// TIA Portal V16 export
// export: Created 2021-12-01T20:36:48.810046Z, ExportSetting WithDefaults, DisplayName Totally Integrated Automation Portal, DisplayVersion V16 Update 4, DisplayName TIA Portal Version Control Interface, DisplayVersion V16 Update 2, DisplayName TIA Portal Openness, DisplayVersion V16 Update 4, DisplayName SINAMICS Startdrive Advanced, DisplayVersion V16 Update 5, DisplayName SINAMICS Startdrive G130, G150, S120, S150, SINAMICS MV, S210, DisplayVersion V16 Update 5, DisplayName SINAMICS Startdrive G110M, G120, G120C, G120D, G120P, G115D, DisplayVersion V16 Update 5, DisplayName STEP 7 Professional, DisplayVersion V16 Update 4, DisplayName STEP 7 Safety, DisplayVersion V16, DisplayName WinCC Advanced, DisplayVersion V16 Update 4
FUNCTION "ST00280_FC" : Void   // FC102, LAD
TITLE = ST00280
{ S7_Optimized_Access := 'TRUE' }
VERSION : 0.1
// stored: AutoNumber true, IsIECCheckEnabled false, SetENOAutomatically false, UDAEnableTagReadback false
   VAR_IN_OUT
      OPMODE : "OPMODE_OUT_UDT";
      HMI_EXTENSION : "HMI_EXTENSION_PANEL_UDT";
   END_VAR
   VAR_TEMP
      EmptyHS : "RT_HANDSHAKE_UDT";
   END_VAR
BEGIN

REGION Network 1: Alarm
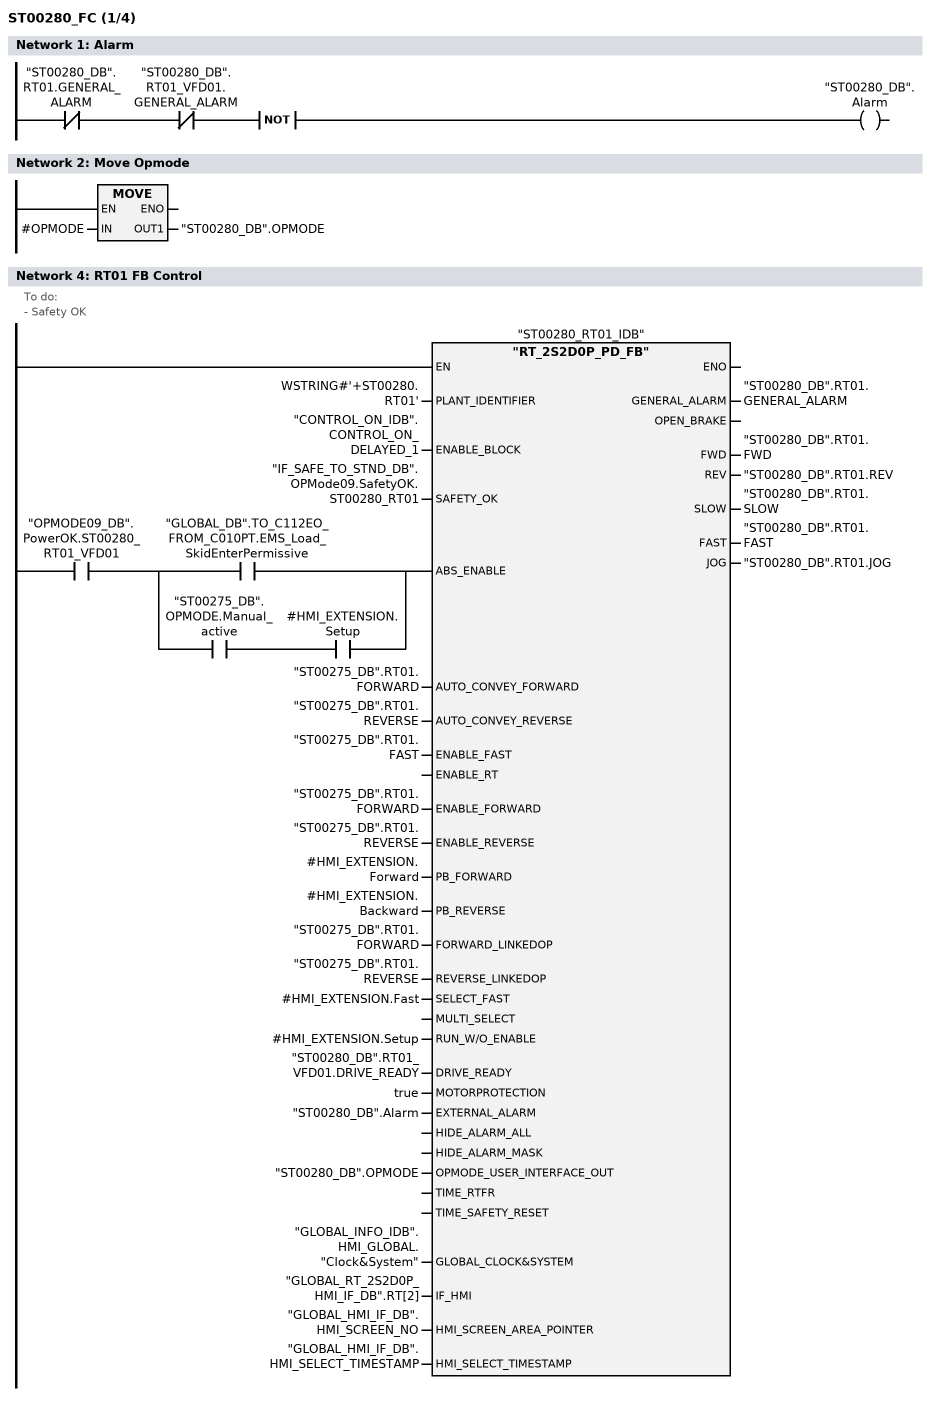
   RUNG wire#powerrail
      I_Contact( "ST00280_DB".RT01.GENERAL_ALARM )
      I_Contact( "ST00280_DB".RT01_VFD01.GENERAL_ALARM )
      Not()
      Coil( "ST00280_DB".Alarm )
   END_RUNG
   // the same network as SCL:
   "ST00280_DB".Alarm := NOT (NOT "ST00280_DB".RT01.GENERAL_ALARM AND NOT "ST00280_DB".RT01_VFD01.GENERAL_ALARM);
END_REGION

REGION Network 2: Move Opmode
   RUNG wire#powerrail
      Move(in := #OPMODE, out1 => "ST00280_DB".OPMODE)
   END_RUNG
   // the same network as SCL:
   "ST00280_DB".OPMODE := #OPMODE;
END_REGION

REGION Network 3: *******************RT01 Control*******************
END_REGION

REGION Network 4: RT01 FB Control
   // To do:
   // 										- Safety OK
   RUNG wire#powerrail
      "ST00280_RT01_IDB"(ABS_ENABLE := wire#w2, PLANT_IDENTIFIER := WSTRING#'+ST00280.RT01', ENABLE_BLOCK := "CONTROL_ON_IDB".CONTROL_ON_DELAYED_1, SAFETY_OK := "IF_SAFE_TO_STND_DB".OPMode09.SafetyOK.ST00280_RT01, AUTO_CONVEY_FORWARD := "ST00275_DB".RT01.FORWARD, AUTO_CONVEY_REVERSE := "ST00275_DB".RT01.REVERSE, ENABLE_FAST := "ST00275_DB".RT01.FAST, ENABLE_RT :=, ENABLE_FORWARD := "ST00275_DB".RT01.FORWARD, ENABLE_REVERSE := "ST00275_DB".RT01.REVERSE, PB_FORWARD := #HMI_EXTENSION.Forward, PB_REVERSE := #HMI_EXTENSION.Backward, FORWARD_LINKEDOP := "ST00275_DB".RT01.FORWARD, REVERSE_LINKEDOP := "ST00275_DB".RT01.REVERSE, SELECT_FAST := #HMI_EXTENSION.Fast, MULTI_SELECT :=, "RUN_W/O_ENABLE" := #HMI_EXTENSION.Setup, DRIVE_READY := "ST00280_DB".RT01_VFD01.DRIVE_READY, MOTORPROTECTION := true, EXTERNAL_ALARM := "ST00280_DB".Alarm, HIDE_ALARM_ALL :=, HIDE_ALARM_MASK :=, OPMODE_USER_INTERFACE_OUT := "ST00280_DB".OPMODE, TIME_RTFR :=, TIME_SAFETY_RESET :=, "GLOBAL_CLOCK&SYSTEM" := "GLOBAL_INFO_IDB".HMI_GLOBAL."Clock&System", IF_HMI := "GLOBAL_RT_2S2D0P_HMI_IF_DB".RT[2], HMI_SCREEN_AREA_POINTER := "GLOBAL_HMI_IF_DB".HMI_SCREEN_NO, HMI_SELECT_TIMESTAMP := "GLOBAL_HMI_IF_DB".HMI_SELECT_TIMESTAMP, GENERAL_ALARM => "ST00280_DB".RT01.GENERAL_ALARM, OPEN_BRAKE =>, FWD => "ST00280_DB".RT01.FWD, REV => "ST00280_DB".RT01.REV, SLOW => "ST00280_DB".RT01.SLOW, FAST => "ST00280_DB".RT01.FAST, JOG => "ST00280_DB".RT01.JOG)
   END_RUNG
   RUNG wire#powerrail
      Contact( "OPMODE09_DB".PowerOK.ST00280_RT01_VFD01 )
      wire#w1
      Contact( "GLOBAL_DB".TO_C112EO_FROM_C010PT.EMS_Load_SkidEnterPermissive )
   END_RUNG wire#w2
   RUNG wire#w1
      Contact( "ST00275_DB".OPMODE.Manual_active )
      Contact( #HMI_EXTENSION.Setup )
   END_RUNG wire#w2
   // the same network as SCL:
   "ST00280_RT01_IDB"(PLANT_IDENTIFIER := WSTRING#'+ST00280.RT01',   // "RT_2S2D0P_PD_FB"
                      ENABLE_BLOCK := "CONTROL_ON_IDB".CONTROL_ON_DELAYED_1,
                      SAFETY_OK := "IF_SAFE_TO_STND_DB".OPMode09.SafetyOK.ST00280_RT01,
                      ABS_ENABLE := "OPMODE09_DB".PowerOK.ST00280_RT01_VFD01 AND ("GLOBAL_DB".TO_C112EO_FROM_C010PT.EMS_Load_SkidEnterPermissive OR ("ST00275_DB".OPMODE.Manual_active AND #HMI_EXTENSION.Setup)),
                      AUTO_CONVEY_FORWARD := "ST00275_DB".RT01.FORWARD,
                      AUTO_CONVEY_REVERSE := "ST00275_DB".RT01.REVERSE,
                      ENABLE_FAST := "ST00275_DB".RT01.FAST,
                      ENABLE_FORWARD := "ST00275_DB".RT01.FORWARD,
                      ENABLE_REVERSE := "ST00275_DB".RT01.REVERSE,
                      PB_FORWARD := #HMI_EXTENSION.Forward,
                      PB_REVERSE := #HMI_EXTENSION.Backward,
                      FORWARD_LINKEDOP := "ST00275_DB".RT01.FORWARD,
                      REVERSE_LINKEDOP := "ST00275_DB".RT01.REVERSE,
                      SELECT_FAST := #HMI_EXTENSION.Fast,
                      "RUN_W/O_ENABLE" := #HMI_EXTENSION.Setup,
                      DRIVE_READY := "ST00280_DB".RT01_VFD01.DRIVE_READY,
                      MOTORPROTECTION := true,
                      EXTERNAL_ALARM := "ST00280_DB".Alarm,
                      OPMODE_USER_INTERFACE_OUT := "ST00280_DB".OPMODE,
                      "GLOBAL_CLOCK&SYSTEM" := "GLOBAL_INFO_IDB".HMI_GLOBAL."Clock&System",
                      IF_HMI := "GLOBAL_RT_2S2D0P_HMI_IF_DB".RT[2],
                      HMI_SCREEN_AREA_POINTER := "GLOBAL_HMI_IF_DB".HMI_SCREEN_NO,
                      HMI_SELECT_TIMESTAMP := "GLOBAL_HMI_IF_DB".HMI_SELECT_TIMESTAMP,
                      GENERAL_ALARM => "ST00280_DB".RT01.GENERAL_ALARM,
                      FWD => "ST00280_DB".RT01.FWD,
                      REV => "ST00280_DB".RT01.REV,
                      SLOW => "ST00280_DB".RT01.SLOW,
                      FAST => "ST00280_DB".RT01.FAST,
                      JOG => "ST00280_DB".RT01.JOG);
END_REGION

REGION Network 5: RT01 Speed
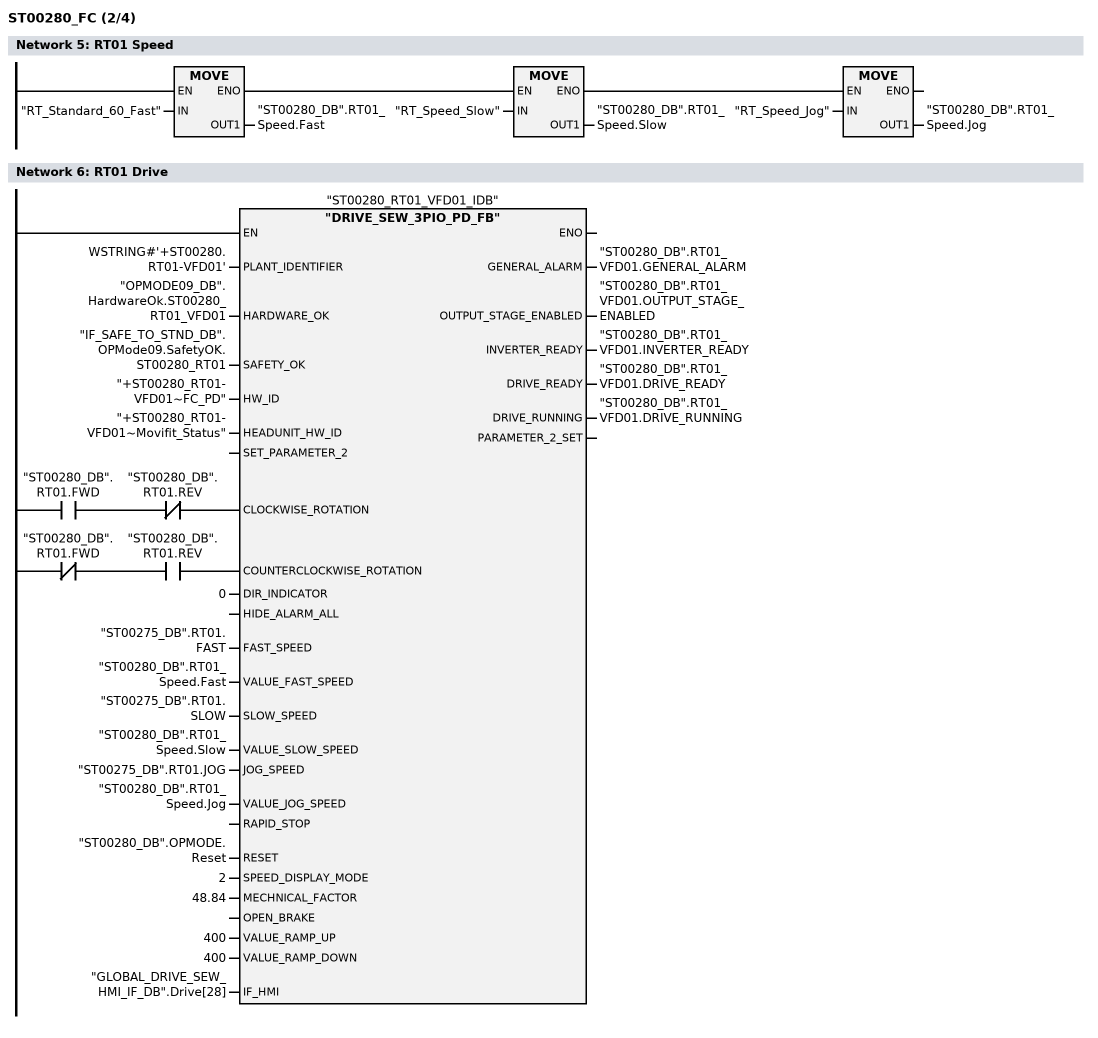
   RUNG wire#powerrail
      Move(in := "RT_Standard_60_Fast", out1 => "ST00280_DB".RT01_Speed.Fast)
      Move(in := "RT_Speed_Slow", out1 => "ST00280_DB".RT01_Speed.Slow)
      Move(in := "RT_Speed_Jog", out1 => "ST00280_DB".RT01_Speed.Jog)
   END_RUNG
   // the same network as SCL:
   "ST00280_DB".RT01_Speed.Fast := "RT_Standard_60_Fast";
   "ST00280_DB".RT01_Speed.Slow := "RT_Speed_Slow";
   "ST00280_DB".RT01_Speed.Jog := "RT_Speed_Jog";
END_REGION

REGION Network 6: RT01 Drive
   RUNG wire#powerrail
      "ST00280_RT01_VFD01_IDB"(CLOCKWISE_ROTATION := wire#w1, COUNTERCLOCKWISE_ROTATION := wire#w2, PLANT_IDENTIFIER := WSTRING#'+ST00280.RT01-VFD01', HARDWARE_OK := "OPMODE09_DB".HardwareOk.ST00280_RT01_VFD01, SAFETY_OK := "IF_SAFE_TO_STND_DB".OPMode09.SafetyOK.ST00280_RT01, HW_ID := "+ST00280_RT01-VFD01~FC_PD", HEADUNIT_HW_ID := "+ST00280_RT01-VFD01~Movifit_Status", SET_PARAMETER_2 :=, DIR_INDICATOR := 0, HIDE_ALARM_ALL :=, FAST_SPEED := "ST00275_DB".RT01.FAST, VALUE_FAST_SPEED := "ST00280_DB".RT01_Speed.Fast, SLOW_SPEED := "ST00275_DB".RT01.SLOW, VALUE_SLOW_SPEED := "ST00280_DB".RT01_Speed.Slow, JOG_SPEED := "ST00275_DB".RT01.JOG, VALUE_JOG_SPEED := "ST00280_DB".RT01_Speed.Jog, RAPID_STOP :=, RESET := "ST00280_DB".OPMODE.Reset, SPEED_DISPLAY_MODE := 2, MECHNICAL_FACTOR := 48.84, OPEN_BRAKE :=, VALUE_RAMP_UP := 400, VALUE_RAMP_DOWN := 400, IF_HMI := "GLOBAL_DRIVE_SEW_HMI_IF_DB".Drive[28], GENERAL_ALARM => "ST00280_DB".RT01_VFD01.GENERAL_ALARM, OUTPUT_STAGE_ENABLED => "ST00280_DB".RT01_VFD01.OUTPUT_STAGE_ENABLED, INVERTER_READY => "ST00280_DB".RT01_VFD01.INVERTER_READY, DRIVE_READY => "ST00280_DB".RT01_VFD01.DRIVE_READY, DRIVE_RUNNING => "ST00280_DB".RT01_VFD01.DRIVE_RUNNING, PARAMETER_2_SET =>)
   END_RUNG
   RUNG wire#powerrail
      Contact( "ST00280_DB".RT01.FWD )
      I_Contact( "ST00280_DB".RT01.REV )
   END_RUNG wire#w1
   RUNG wire#powerrail
      I_Contact( "ST00280_DB".RT01.FWD )
      Contact( "ST00280_DB".RT01.REV )
   END_RUNG wire#w2
   // the same network as SCL:
   "ST00280_RT01_VFD01_IDB"(PLANT_IDENTIFIER := WSTRING#'+ST00280.RT01-VFD01',   // "DRIVE_SEW_3PIO_PD_FB"
                           HARDWARE_OK := "OPMODE09_DB".HardwareOk.ST00280_RT01_VFD01,
                           SAFETY_OK := "IF_SAFE_TO_STND_DB".OPMode09.SafetyOK.ST00280_RT01,
                           HW_ID := "+ST00280_RT01-VFD01~FC_PD",
                           HEADUNIT_HW_ID := "+ST00280_RT01-VFD01~Movifit_Status",
                           CLOCKWISE_ROTATION := "ST00280_DB".RT01.FWD AND NOT "ST00280_DB".RT01.REV,
                           COUNTERCLOCKWISE_ROTATION := NOT "ST00280_DB".RT01.FWD AND "ST00280_DB".RT01.REV,
                           DIR_INDICATOR := 0,
                           FAST_SPEED := "ST00275_DB".RT01.FAST,
                           VALUE_FAST_SPEED := "ST00280_DB".RT01_Speed.Fast,
                           SLOW_SPEED := "ST00275_DB".RT01.SLOW,
                           VALUE_SLOW_SPEED := "ST00280_DB".RT01_Speed.Slow,
                           JOG_SPEED := "ST00275_DB".RT01.JOG,
                           VALUE_JOG_SPEED := "ST00280_DB".RT01_Speed.Jog,
                           RESET := "ST00280_DB".OPMODE.Reset,
                           SPEED_DISPLAY_MODE := 2,
                           MECHNICAL_FACTOR := 48.84,
                           VALUE_RAMP_UP := 400,
                           VALUE_RAMP_DOWN := 400,
                           IF_HMI := "GLOBAL_DRIVE_SEW_HMI_IF_DB".Drive[28],
                           GENERAL_ALARM => "ST00280_DB".RT01_VFD01.GENERAL_ALARM,
                           OUTPUT_STAGE_ENABLED => "ST00280_DB".RT01_VFD01.OUTPUT_STAGE_ENABLED,
                           INVERTER_READY => "ST00280_DB".RT01_VFD01.INVERTER_READY,
                           DRIVE_READY => "ST00280_DB".RT01_VFD01.DRIVE_READY,
                           DRIVE_RUNNING => "ST00280_DB".RT01_VFD01.DRIVE_RUNNING);
END_REGION

REGION Network 7: *******************PO01 Control*******************
END_REGION

REGION Network 8 (SCL): PO01 Parameters
   "ST00280_DB".PO01.PARA_SET.Para.PosEndForward2 := false;
   "ST00280_DB".PO01.PARA_SET.Para.PosEndReverse2 := false;

   "ST00280_DB".PO01.PARA_SET.Set.SetRT := 100;
   "ST00280_DB".PO01.PARA_SET.Set.TimePosLeft := 10;
END_REGION

REGION Network 9: PO01 FB Control
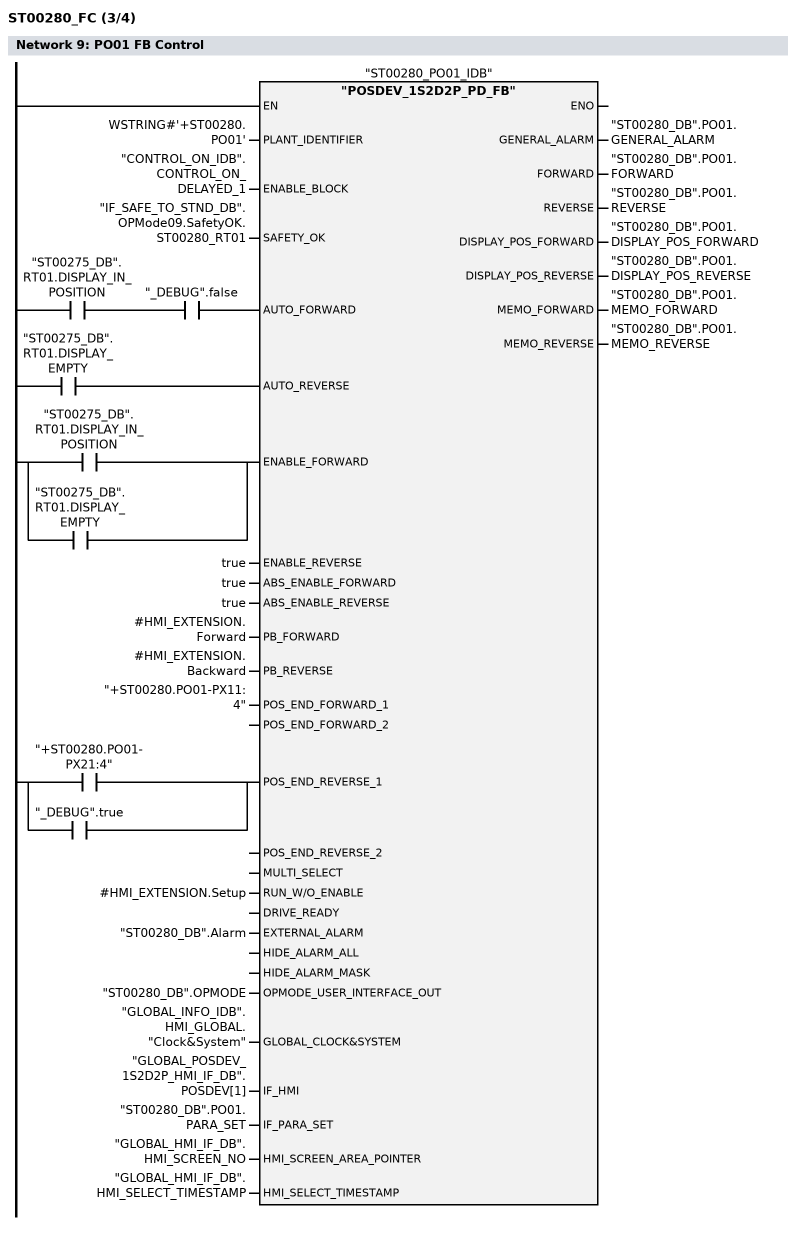
   RUNG wire#powerrail
      "ST00280_PO01_IDB"(AUTO_FORWARD := wire#w1, AUTO_REVERSE := wire#w2, ENABLE_FORWARD := wire#w3, POS_END_REVERSE_1 := wire#w4, PLANT_IDENTIFIER := WSTRING#'+ST00280.PO01', ENABLE_BLOCK := "CONTROL_ON_IDB".CONTROL_ON_DELAYED_1, SAFETY_OK := "IF_SAFE_TO_STND_DB".OPMode09.SafetyOK.ST00280_RT01, ENABLE_REVERSE := true, ABS_ENABLE_FORWARD := true, ABS_ENABLE_REVERSE := true, PB_FORWARD := #HMI_EXTENSION.Forward, PB_REVERSE := #HMI_EXTENSION.Backward, POS_END_FORWARD_1 := "+ST00280.PO01-PX11:4", POS_END_FORWARD_2 :=, POS_END_REVERSE_2 :=, MULTI_SELECT :=, "RUN_W/O_ENABLE" := #HMI_EXTENSION.Setup, DRIVE_READY :=, EXTERNAL_ALARM := "ST00280_DB".Alarm, HIDE_ALARM_ALL :=, HIDE_ALARM_MASK :=, OPMODE_USER_INTERFACE_OUT := "ST00280_DB".OPMODE, "GLOBAL_CLOCK&SYSTEM" := "GLOBAL_INFO_IDB".HMI_GLOBAL."Clock&System", IF_HMI := "GLOBAL_POSDEV_1S2D2P_HMI_IF_DB".POSDEV[1], IF_PARA_SET := "ST00280_DB".PO01.PARA_SET, HMI_SCREEN_AREA_POINTER := "GLOBAL_HMI_IF_DB".HMI_SCREEN_NO, HMI_SELECT_TIMESTAMP := "GLOBAL_HMI_IF_DB".HMI_SELECT_TIMESTAMP, GENERAL_ALARM => "ST00280_DB".PO01.GENERAL_ALARM, FORWARD => "ST00280_DB".PO01.FORWARD, REVERSE => "ST00280_DB".PO01.REVERSE, DISPLAY_POS_FORWARD => "ST00280_DB".PO01.DISPLAY_POS_FORWARD, DISPLAY_POS_REVERSE => "ST00280_DB".PO01.DISPLAY_POS_REVERSE, MEMO_FORWARD => "ST00280_DB".PO01.MEMO_FORWARD, MEMO_REVERSE => "ST00280_DB".PO01.MEMO_REVERSE)
   END_RUNG
   RUNG wire#powerrail
      Contact( "ST00275_DB".RT01.DISPLAY_IN_POSITION )
      Contact( "_DEBUG".false )
   END_RUNG wire#w1
   RUNG wire#powerrail
      Contact( "ST00275_DB".RT01.DISPLAY_EMPTY )
   END_RUNG wire#w2
   RUNG wire#powerrail
      Contact( "ST00275_DB".RT01.DISPLAY_IN_POSITION )
   END_RUNG wire#w3
   RUNG wire#powerrail
      Contact( "ST00275_DB".RT01.DISPLAY_EMPTY )
   END_RUNG wire#w3
   RUNG wire#powerrail
      Contact( "+ST00280.PO01-PX21:4" )
   END_RUNG wire#w4
   RUNG wire#powerrail
      Contact( "_DEBUG".true )
   END_RUNG wire#w4
   // the same network as SCL:
   "ST00280_PO01_IDB"(PLANT_IDENTIFIER := WSTRING#'+ST00280.PO01',   // "POSDEV_1S2D2P_PD_FB"
                      ENABLE_BLOCK := "CONTROL_ON_IDB".CONTROL_ON_DELAYED_1,
                      SAFETY_OK := "IF_SAFE_TO_STND_DB".OPMode09.SafetyOK.ST00280_RT01,
                      AUTO_FORWARD := "ST00275_DB".RT01.DISPLAY_IN_POSITION AND "_DEBUG".false,
                      AUTO_REVERSE := "ST00275_DB".RT01.DISPLAY_EMPTY,
                      ENABLE_FORWARD := "ST00275_DB".RT01.DISPLAY_IN_POSITION OR "ST00275_DB".RT01.DISPLAY_EMPTY,
                      ENABLE_REVERSE := true,
                      ABS_ENABLE_FORWARD := true,
                      ABS_ENABLE_REVERSE := true,
                      PB_FORWARD := #HMI_EXTENSION.Forward,
                      PB_REVERSE := #HMI_EXTENSION.Backward,
                      POS_END_FORWARD_1 := "+ST00280.PO01-PX11:4",
                      POS_END_REVERSE_1 := "+ST00280.PO01-PX21:4" OR "_DEBUG".true,
                      "RUN_W/O_ENABLE" := #HMI_EXTENSION.Setup,
                      EXTERNAL_ALARM := "ST00280_DB".Alarm,
                      OPMODE_USER_INTERFACE_OUT := "ST00280_DB".OPMODE,
                      "GLOBAL_CLOCK&SYSTEM" := "GLOBAL_INFO_IDB".HMI_GLOBAL."Clock&System",
                      IF_HMI := "GLOBAL_POSDEV_1S2D2P_HMI_IF_DB".POSDEV[1],
                      IF_PARA_SET := "ST00280_DB".PO01.PARA_SET,
                      HMI_SCREEN_AREA_POINTER := "GLOBAL_HMI_IF_DB".HMI_SCREEN_NO,
                      HMI_SELECT_TIMESTAMP := "GLOBAL_HMI_IF_DB".HMI_SELECT_TIMESTAMP,
                      GENERAL_ALARM => "ST00280_DB".PO01.GENERAL_ALARM,
                      FORWARD => "ST00280_DB".PO01.FORWARD,
                      REVERSE => "ST00280_DB".PO01.REVERSE,
                      DISPLAY_POS_FORWARD => "ST00280_DB".PO01.DISPLAY_POS_FORWARD,
                      DISPLAY_POS_REVERSE => "ST00280_DB".PO01.DISPLAY_POS_REVERSE,
                      MEMO_FORWARD => "ST00280_DB".PO01.MEMO_FORWARD,
                      MEMO_REVERSE => "ST00280_DB".PO01.MEMO_REVERSE);
END_REGION

REGION Network 10: PO01 Output control
   // To Do: connect position signals
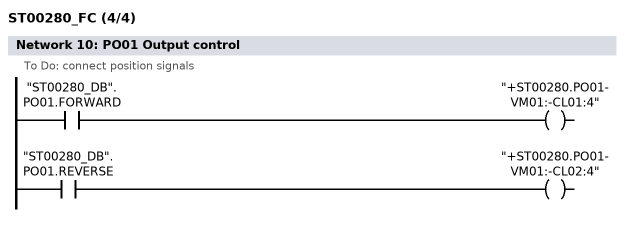
   RUNG wire#powerrail
      Contact( "ST00280_DB".PO01.FORWARD )
      Coil( "+ST00280.PO01-VM01:-CL01:4" )
   END_RUNG
   RUNG wire#powerrail
      Contact( "ST00280_DB".PO01.REVERSE )
      Coil( "+ST00280.PO01-VM01:-CL02:4" )
   END_RUNG
   // the same network as SCL:
   "+ST00280.PO01-VM01:-CL01:4" := "ST00280_DB".PO01.FORWARD;
   "+ST00280.PO01-VM01:-CL02:4" := "ST00280_DB".PO01.REVERSE;
END_REGION
END_FUNCTION
